FUNCTION_BLOCK FB_LevelControl
VAR_INPUT
END_VAR
VAR_OUTPUT
END_VAR
VAR
	byH: BOOL;
	byL: BOOL;
	buL: BOOL;
	fbReactorUpperLimit: FB_LimitSwitch;
	fbReactorLowerLimit: FB_LimitSwitch;
END_VAR

(*//Level Control state
IF HMI.bLevelControlSwitch = 1 THEN
	HMI.sLevelControlState := 'AUTO';
END_IF
IF HMI.bLevelControlSwitch = 0 THEN
	HMI.sLevelControlState := 'MAN';
END_IF
//Level Valve state
IF IO.bReactorLu = 1 THEN
	HMI.sLevelValveState := 'CLOSE';
END_IF
IF IO.bReactorLu = 0 THEN
	HMI.sLevelValveState := 'OPEN';
END_IF

//Read measurement values
// Level
byH := IO.bReactorHy;
byL := IO.bReactorLy;
buL := IO.bReactorLu;

IF HMI.bLevelControlSwitch THEN
	fbReactorUpperLimit(I_LimitSwitch := IO.bReactorHy, I_LowerLimit := FALSE, I_AlarmTimeSecs := 3);
	fbReactorLowerLimit(I_LimitSwitch := IO.bReactorLy, I_LowerLimit := TRUE, I_AlarmTimeSecs := 1);
	IF fbReactorUpperLimit.O_LimitAlarm THEN
		IO.bReactorLu := TRUE;
	END_IF
	IF fbReactorLowerLimit.O_LimitAlarm THEN
		IO.bReactorLu := FALSE;
	END_IF
END_IF

//IF fbReactorUpperLimit.O_LimitAlarm THEN

//Auto Control
(*IF HMI.bLevelControlSwitch THEN
	IF byL = 0 THEN
		IF IO.bReactorLu = 1 THEN
			IO.bReactorLu := 0;
		END_IF
	ELSIF byH = 1 THEN
		IF IO.bReactorLu = 0 THEN
			IO.bReactorLu := 1;
		END_IF
	// exit auto mode when filling 
	(*ELSIF byL = 0 AND byH = 0 THEN
		HMI.bLevelControlSwitch := 0;*)
	END_IF
END_IF*)
*)

END_FUNCTION_BLOCK

(* stored: Version 1.1.0.1, ProductVersion 3.1.4024.9
   POU FB_LevelControl: Id {32cd3e91-9b01-412d-a1bd-2ea8d1d450bf}, SpecialFunc None *)
